// {attribute 'qualified_only'}
// {attribute 'strict'}
// {attribute 'to_string'}
TYPE MoveState_t :
(
	MOVESTATE_INIT,
	MOVESTATE_ENABLE,
	MOVESTATE_IDLE,
	MOVESTATE_FORWARD,
	MOVESTATE_BACKWARDS,
	MOVESTATE_HALT,
	MOVESTATE_BACKWARDSSLOW,
	MOVESTATE_NEWTARGETPOSITION,
	MOVESTATE_ERROR,
	MOVESTATE_RESET
) UDINT;
END_TYPE

(* stored: Version 1.1.0.1
   DUT MoveState_t: Id {79e54ced-6f77-485e-ad33-7ba47d76694a} *)
